FUNCTION_BLOCK OperatorArithmetic (* Template for an empty basic function block *)
  (* Standard: 61499-2; Description: Copyright (c) 2019 Jan Holzweber This program and the accompanying materials are made available under the terms of the Eclipse Public License 2.0 which is available at https://www.eclipse.org/legal/epl-2.0/ SPDX-License-Identifier: EPL-2.0 *)
  (* Version 1.0, 2019-06-05, jholz *)
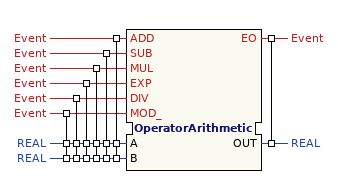
  EVENT_INPUT
    ADD WITH A, B;
    SUB WITH A, B;
    MUL WITH A, B;
    EXP WITH A, B;
    DIV WITH A, B;
    MOD_ WITH A, B;
  END_EVENT
  EVENT_OUTPUT
    EO WITH OUT;
  END_EVENT
  VAR_INPUT
    A : REAL;
    B : REAL;
  END_VAR
  VAR_OUTPUT
    OUT : REAL;
  END_VAR
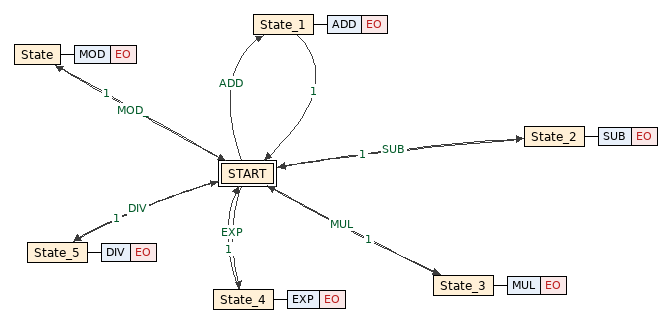
  EC_STATES
    START; (* Initial State *)
    State : MOD -> EO;
    State_1 : ADD -> EO;
    State_2 : SUB -> EO;
    State_3 : MUL -> EO;
    State_4 : EXP -> EO;
    State_5 : DIV -> EO;
  END_STATES
  EC_TRANSITIONS
    State_1 TO START := 1;
    START TO State_1 := ADD;
    START TO State_2 := SUB;
    START TO State_3 := MUL;
    START TO State_4 := EXP;
    START TO State_5 := DIV;
    START TO State := MOD_;
    State TO START := 1;
    State_5 TO START := 1;
    State_4 TO START := 1;
    State_3 TO START := 1;
    State_2 TO START := 1;
  END_TRANSITIONS
  ALGORITHM ADD IN ST: (* new algorithm *)
OUT:=A+B;
  END_ALGORITHM
  ALGORITHM SUB IN ST: (* new algorithm *)
OUT:=A-B;
  END_ALGORITHM
  ALGORITHM MUL IN ST: (* new algorithm *)
OUT:=A*B;
  END_ALGORITHM
  ALGORITHM EXP IN ST: (* new algorithm *)
OUT:=A**B;
  END_ALGORITHM
  ALGORITHM DIV IN ST: (* new algorithm *)
OUT:=A / B;
  END_ALGORITHM
  ALGORITHM MOD IN ST: (* new algorithm *)
OUT:=A MOD B;
  END_ALGORITHM
END_FUNCTION_BLOCK
